TYPE ST_Camera :
STRUCT
	
	State								: E_Camera_State;
	CMD									: ST_GeneralStationCMD;
	Status								: ST_StationStatus;

END_STRUCT
END_TYPE

(* stored: Version 1.1.0.1, ProductVersion 3.1.4024.13
   DUT ST_Camera: Id {cf904a9d-85be-4d55-8b2c-a8b096053ffe} *)
